// TwinCAT 3 PLC project PLC
// ProgramVersion: 3.1.4024.0
// libraries:
//   Tc2_ControllerToolbox, * (Beckhoff Automation GmbH)
//   Tc2_Standard, * (Beckhoff Automation GmbH)
//   Tc2_System, * (Beckhoff Automation GmbH)
//   Tc3_Module, * (Beckhoff Automation GmbH)
//   TcUnit, * (www.tcunit.org)
// project tree:
//   / PlcTask.TcTTO
//   POUs/3DOF robot/ FB_Clamp_INT.TcPOU, FB_RC_Servo.TcPOU, FB_Sequence_Executor.TcPOU, FB_Sequence_Recorder.TcPOU
//   POUs/3DOF robot/TEST/ FB_Clamp_INT_Test.TcPOU, FB_RC_Servo_Test.TcPOU, FB_Sequence_Recorder_Test.TcPOU, PRG_TEST_ThreeDOF_robot.TcPOU
//   POUs/Controller/ FB_Adaptive_PID_Controller.TcPOU, FB_Hysteresis.TcPOU, FB_PID_Controller.TcPOU
//   POUs/Controller/TEST/ PRG_Controller_TEST.TcPOU
//   POUs/Equipment simulation/ FB_MassSpringDamper.TcPOU, FB_Tank.TcPOU
//   POUs/Equipment simulation/TEST/ PRG_EquipmentSimulation_TEST.TcPOU
//   POUs/Filters/ FB_Filter_Floating_Average.TcPOU, FB_Filter_HighPass.TcPOU, FB_Filter_LowPass.TcPOU
//   POUs/Filters/TEST/ PRG_Filters_TEST.TcPOU
//   POUs/ Notes.TcPOU, Tips_and_tricks.TcPOU
//   POUs/Signal generators/ FB_Generator_PWM.TcPOU, FB_Generator_Random.TcPOU, FB_Generator_Sawtooth.TcPOU, FB_Generator_Sine.TcPOU, FB_Generator_Square.TcPOU, FB_Generator_Triangular.TcPOU
//   POUs/Signal generators/TEST/ PRG_SignalGenerators_TEST.TcPOU
//   POUs/Unit test example/ FB_Max_Value.TcPOU, FB_Max_Value_Test.TcPOU, PRG_TEST.TcPOU
// real-time tasks:
//   TASK PlcTask: cycle T#10ms, priority 20, ADS port 350

CONFIGURATION PLC
    RESOURCE PLC ON TwinCAT3
        TASK PlcTask(INTERVAL := T#10ms, PRIORITY := 20);
        PROGRAM PRG_TEST_ThreeDOF_robot WITH PlcTask : PRG_TEST_ThreeDOF_robot;
    END_RESOURCE
END_CONFIGURATION

// ---- POUs/3DOF robot/TEST/PRG_TEST_ThreeDOF_robot.TcPOU
PROGRAM PRG_TEST_ThreeDOF_robot
VAR
	fb_RC_Servo_Test : FB_RC_Servo_Test;
	fb_Sequence_Recorder : FB_Sequence_Recorder_Test;
	fb_Clamp_INT_Test : FB_Clamp_INT_Test;
END_VAR

TcUnit.RUN();

END_PROGRAM

// ---- POUs/3DOF robot/TEST/FB_RC_Servo_Test.TcPOU
FUNCTION_BLOCK FB_RC_Servo_Test EXTENDS TcUnit.FB_TestSuite

// SetpointReached();
// Stop();

METHOD PRIVATE OutputRamped
VAR_INPUT
END_VAR
END_METHOD

METHOD PRIVATE SetpointChanged
VAR_INPUT
END_VAR
END_METHOD

METHOD SetpointReached
VAR
	Servo : FB_RC_Servo;
	Setpoint : INT := 10;
	ExpectedSetpointReached : INT := 10;
	Result : INT;
END_VAR
TEST('TEST: Setpoint reached');

Servo(stop := FALSE,
	setpoint := Setpoint,
	rampSpeed := 10,
	trapezoidalProfileActive := FALSE,
	servoAngleMin := 0,
	servoAngleMax := 100,
	rampCycleTime := T#1MS,
	currentPositionSetpoint => Result);
	


AssertEquals(Expected := ExpectedSetpointReached,
	Actual := Servo.currentPositionSetpoint,
	Message := 'Expected value not reached');

TEST_FINISHED();
END_METHOD

METHOD PRIVATE StartingPosition
VAR_INPUT
END_VAR
END_METHOD

METHOD PRIVATE Stop
VAR
	stop : BOOL;
	init1 : BOOL := TRUE;
	init2 : BOOL := TRUE;
	init3 : BOOL := TRUE;
	intermediateVal1 : INT;
	intermediateVal2 : INT;
	valuesAreEqualAndNotZero : BOOL := FALSE;
	startValue : INT := 0;
	setpoint : INT := 10000;
	minValue : INT := 0;
	maxValue : INT := 10000;
	cycleTime : TIME := T#1MS;
	rampSpeed : INT := 20;
	FB_Servo: FB_RC_Servo;
	timer1: TON;
	timer2: TON;
	ExpectedValue : BOOL := TRUE;
END_VAR
IF init1 THEN
	stop := FALSE;
	init1 := FALSE;
END_IF;

timer1(IN:= TRUE, PT:= T#1000S, Q=> , ET=> );
timer2(IN:= TRUE, PT:= T#1000S, Q=> , ET=> );

FB_Servo(
	stop:= stop, 
	setpoint:= setpoint, 
	rampSpeed:= rampSpeed, 
	trapezoidalProfileActive:= FALSE, 
	servoAngleMin:= minValue, 
	servoAngleMax:= maxValue, 
	rampCycleTime:= cycleTime, 
	rampStartPos:= startValue, 
	currentPositionSetpoint=> , 
	error=> );

IF timer1.ET > T#1S AND init2 THEN
	stop := TRUE;
	intermediateVal1 := FB_Servo.currentPositionSetpoint;
	init2 := FALSE;
END_IF

IF timer2.ET > T#2S AND init3 THEN
	IF intermediateVal1 = intermediateVal2 AND intermediateVal1 <> 0 THEN
		valuesAreEqualAndNotZero := TRUE;
	END_IF
END_IF

AssertEquals(
Expected:= ExpectedValue,
 Actual:= valuesAreEqualAndNotZero,
 Message:= 'Ramp was not stopped or value was not ramped');
END_METHOD

METHOD PRIVATE Trapezoidal
VAR_INPUT
END_VAR
END_METHOD

END_FUNCTION_BLOCK

// ---- POUs/3DOF robot/FB_RC_Servo.TcPOU
FUNCTION_BLOCK FB_RC_Servo
VAR_INPUT
	stop : BOOL; // Stops motor at current position
	setpoint : INT; // Angle to reach
	rampSpeed : REAL; // Speed setpoint for servo angle
	trapezoidalProfileActive : BOOL; // Smooths speed of servo at start and end of movement
	servoAngleMin : INT; // Lower limit of function block output angle
	servoAngleMax : INT; // Upper limit of function block output angle
	rampCycleTime : TIME; // Set rampCycleTime to the same as the task sycle time
	rampStartPos : INT; // Starting position
END_VAR
VAR_OUTPUT
	currentPositionSetpoint : INT; // The actual output of function block
	error : STRING; // Error output for debug
END_VAR
VAR
	ramp : FB_CTRL_RAMP_GENERATOR;
	rampParameters : ST_CTRL_RAMP_GENERATOR_PARAMS;
END_VAR

rampParameters.fVeloNeg := rampSpeed;
rampParameters.fVeloPos := rampSpeed;
rampParameters.tCtrlCycleTime := rampCycleTime;
rampParameters.tTaskCycleTime := rampCycleTime;
ramp.fStart := rampStartPos;
ramp.fTarget := setpoint;

IF stop THEN
	ramp.bEnable := FALSE;
ELSE
	ramp.bEnable := TRUE;
END_IF

ramp(stParams := rampParameters);

END_FUNCTION_BLOCK

// ---- POUs/3DOF robot/FB_Sequence_Recorder.TcPOU
FUNCTION_BLOCK FB_Sequence_Recorder
VAR_INPUT
	inputBase : INT; // Base angle to be recorded
	inputShoulder : INT; // Shoulder angle to be recorded
	inputElbow : INT; // Elbow angle to be recorded
	recordPosition : BOOL; // Toggle to record current Base, Shoulder, and Elbow angles
	returnPositionAtIndex : INT; // outputBase, outputShoulder, and outputElbow are returned based on this value and recorded positions
	deletePositions : BOOL; // If true, all recorded values will be deleted
END_VAR
VAR_OUTPUT
	outputBase : INT; // Base angle returned based on returnPositonAtIndex
	outputShoulder : INT; // Shoulder angle returned based on returnPositonAtIndex
	outputElbow : INT; // Elbow angle returned based on returnPositonAtIndex
	numberRecordedPositions : INT; // Returns how many positions are saved
	ERROR_arrayFull : BOOL; // Returns true internal storage is full
	ERROR_duplicateValue : BOOL; // Returns true if two duplicate arm positions are attempted recorded simultanously
END_VAR
VAR
	currentIndex : INT := 0;
	basePositions : ARRAY[0..9] OF INT;
	shoulderPositions : ARRAY[0..9] OF INT;
	elbowPositions : ARRAY[0..9] OF INT;
	i : INT;
END_VAR

(* Handle deletion of all positions *)
IF deletePositions THEN
    FOR i := 0 TO 9 DO
        basePositions[i] := 0;
        shoulderPositions[i] := 0;
        elbowPositions[i] := 0;
    END_FOR
    numberRecordedPositions := 0;
    currentIndex := 0;
ELSE
    (* Ensure we do not exceed the array bounds *)
    IF currentIndex >= 10 THEN
        ERROR_arrayFull := TRUE;
    ELSE
        ERROR_arrayFull := FALSE;
        
        (* Check for duplicate only if at least one position is recorded *)
        IF recordPosition AND currentIndex > 0 THEN
            IF basePositions[currentIndex - 1] = inputBase AND 
               shoulderPositions[currentIndex - 1] = inputShoulder AND 
               elbowPositions[currentIndex - 1] = inputElbow THEN
                ERROR_duplicateValue := TRUE;
            ELSE
                ERROR_duplicateValue := FALSE;
            END_IF
        END_IF

        (* Record position if not a duplicate and space is available *)
        IF recordPosition AND NOT ERROR_duplicateValue AND NOT ERROR_arrayFull THEN
            basePositions[currentIndex] := inputBase;
            shoulderPositions[currentIndex] := inputShoulder;
            elbowPositions[currentIndex] := inputElbow;
            currentIndex := currentIndex + 1;
        END_IF
    END_IF

    (* Update the number of recorded positions *)
    numberRecordedPositions := currentIndex;
END_IF;

(* Return recorded position based on the requested index, with bounds check *)
IF returnPositionAtIndex >= 0 AND returnPositionAtIndex < currentIndex THEN
    outputBase := basePositions[returnPositionAtIndex];
    outputShoulder := shoulderPositions[returnPositionAtIndex];
    outputElbow := elbowPositions[returnPositionAtIndex];
ELSE
    outputBase := 0;
    outputShoulder := 0;
    outputElbow := 0;
END_IF;

END_FUNCTION_BLOCK

// ---- POUs/3DOF robot/TEST/FB_Sequence_Recorder_Test.TcPOU
FUNCTION_BLOCK FB_Sequence_Recorder_Test EXTENDS TcUnit.FB_TestSuite

AddOnePosition();
AddTwoPositions();
ClearPositions();
AddTwoClearAddOne();
TryAddDuplicatePosition();
NumberOfPositionsStored();
ZeroPositionsStored();
ArrayFull();

METHOD AddOnePosition
VAR
	inputBaseAngle : INT := 123;
	inputShoulderAngle : INT := 123;
	inputElbowAngle : INT := 123;
	expectedBaseAngle : INT := 123;
	actualBaseAngle : INT;
	FB_Seq_Rec: FB_Sequence_Recorder;
	recordPosition : BOOL := TRUE;
END_VAR
TEST('TEST: Add one position');

FB_Seq_Rec(
	inputBase:= inputBaseAngle, 
	inputShoulder:= inputShoulderAngle, 
	inputElbow:= inputElbowAngle, 
	recordPosition:= recordPosition, 
	returnPositionAtIndex:= 0, 
	deletePositions:= FALSE, 
	outputBase=> actualBaseAngle, 
	outputShoulder=> , 
	outputElbow=> , 
	numberRecordedPositions=> , 
	ERROR_arrayFull=> );

IF recordPosition THEN
	recordPosition := FALSE;
END_IF

AssertEquals(Expected := expectedBaseAngle,
	Actual := actualBaseAngle,
	Message := 'Position 1 was not recorded');
	
TEST_FINISHED();
END_METHOD

METHOD AddTwoClearAddOne
VAR
	inputBaseAngle1 : INT := 123;
	inputShoulderAngle1 : INT := 123;
	inputElbowAngle1 : INT := 123;
	expectedBaseAngle1 : INT := 123;
	inputBaseAngle2 : INT := 234;
	inputShoulderAngle2 : INT := 234;
	inputElbowAngle2 : INT := 234;
	expectedShoulderAngle2 : INT := 234;
	actualShoulderAngle1 : INT;
	actualShoulderAngle2 : INT;
	FB_Seq_Rec: FB_Sequence_Recorder;
	recordPosition : BOOL := TRUE;
	delete : BOOL := FALSE;
END_VAR
TEST('TEST: Add two, delete, then add one position');

FB_Seq_Rec(
	inputBase:= inputBaseAngle1, 
	inputShoulder:= inputShoulderAngle1, 
	inputElbow:= inputElbowAngle1, 
	recordPosition:= recordPosition, 
	returnPositionAtIndex:= 0, 
	deletePositions:= delete, 
	outputBase=> actualShoulderAngle1, 
	outputShoulder=> , 
	outputElbow=> , 
	numberRecordedPositions=> , 
	ERROR_arrayFull=> );
	
FB_Seq_Rec(
	inputBase:= inputBaseAngle2, 
	inputShoulder:= inputShoulderAngle2, 
	inputElbow:= inputElbowAngle2, 
	recordPosition:= recordPosition, 
	returnPositionAtIndex:= 1, 
	deletePositions:= delete, 
	outputBase=> , 
	outputShoulder=> actualShoulderAngle2, 
	outputElbow=> , 
	numberRecordedPositions=> , 
	ERROR_arrayFull=> );

delete := TRUE;
recordPosition := FALSE;

FB_Seq_Rec(
	inputBase:= inputBaseAngle2, 
	inputShoulder:= inputShoulderAngle2, 
	inputElbow:= inputElbowAngle2, 
	recordPosition:= recordPosition, 
	returnPositionAtIndex:= 1, 
	deletePositions:= delete, 
	outputBase=> , 
	outputShoulder=> actualShoulderAngle2, 
	outputElbow=> , 
	numberRecordedPositions=> , 
	ERROR_arrayFull=> );

delete := FALSE;
recordPosition := TRUE;


FB_Seq_Rec(
	inputBase:= inputBaseAngle2, 
	inputShoulder:= inputShoulderAngle2, 
	inputElbow:= inputElbowAngle2, 
	recordPosition:= recordPosition, 
	returnPositionAtIndex:= 0, 
	deletePositions:= delete, 
	outputBase=> , 
	outputShoulder=> actualShoulderAngle2, 
	outputElbow=> , 
	numberRecordedPositions=> , 
	ERROR_arrayFull=> );	

AssertEquals(Expected := expectedShoulderAngle2,
	Actual := actualShoulderAngle2,
	Message := 'Wrong value returned');
	
TEST_FINISHED();
END_METHOD

METHOD AddTwoPositions
VAR
	inputBaseAngle1 : INT := 123;
	inputShoulderAngle1 : INT := 123;
	inputElbowAngle1 : INT := 123;
	expectedBaseAngle1 : INT := 123;
	inputBaseAngle2 : INT := 234;
	inputShoulderAngle2 : INT := 234;
	inputElbowAngle2 : INT := 234;
	expectedShoulderAngle2 : INT := 234;
	actualShoulderAngle1 : INT;
	actualShoulderAngle2 : INT;
	FB_Seq_Rec: FB_Sequence_Recorder;
	recordPosition : BOOL := TRUE;
END_VAR
TEST('TEST: Add two positions');

FB_Seq_Rec(
	inputBase:= inputBaseAngle1, 
	inputShoulder:= inputShoulderAngle1, 
	inputElbow:= inputElbowAngle1, 
	recordPosition:= recordPosition, 
	returnPositionAtIndex:= 0, 
	deletePositions:= FALSE, 
	outputBase=> actualShoulderAngle1, 
	outputShoulder=> , 
	outputElbow=> , 
	numberRecordedPositions=> , 
	ERROR_arrayFull=> );
	
FB_Seq_Rec(
	inputBase:= inputBaseAngle2, 
	inputShoulder:= inputShoulderAngle2, 
	inputElbow:= inputElbowAngle2, 
	recordPosition:= recordPosition, 
	returnPositionAtIndex:= 1, 
	deletePositions:= FALSE, 
	outputBase=> , 
	outputShoulder=> actualShoulderAngle2, 
	outputElbow=> , 
	numberRecordedPositions=> , 
	ERROR_arrayFull=> );

IF recordPosition THEN
	recordPosition := FALSE;
END_IF

AssertEquals(Expected := expectedShoulderAngle2,
	Actual := actualShoulderAngle2,
	Message := 'Position 2 was not recorded');
	
TEST_FINISHED();
END_METHOD

METHOD ArrayFull
VAR
	expectedFeedback : BOOL := TRUE;
	actualFeedback : BOOL;
	FB_Seq_Rec: FB_Sequence_Recorder;
	recordPosition : BOOL := TRUE;
END_VAR
TEST('TEST: Array full');

FB_Seq_Rec(
	inputBase:= 1, 
	inputShoulder:= 0, 
	inputElbow:= 0, 
	recordPosition:= recordPosition, 
	returnPositionAtIndex:= 0, 
	deletePositions:= FALSE, 
	outputBase=> , 
	outputShoulder=> , 
	outputElbow=> , 
	numberRecordedPositions=> , 
	ERROR_arrayFull=> actualFeedback);
	
FB_Seq_Rec(
	inputBase:= 2, 
	inputShoulder:= 0, 
	inputElbow:= 0, 
	recordPosition:= recordPosition, 
	returnPositionAtIndex:= 0, 
	deletePositions:= FALSE, 
	outputBase=> , 
	outputShoulder=> , 
	outputElbow=> , 
	numberRecordedPositions=> , 
	ERROR_arrayFull=> actualFeedback);
	
FB_Seq_Rec(
	inputBase:= 3, 
	inputShoulder:= 0, 
	inputElbow:= 0, 
	recordPosition:= recordPosition, 
	returnPositionAtIndex:= 0, 
	deletePositions:= FALSE, 
	outputBase=> , 
	outputShoulder=> , 
	outputElbow=> , 
	numberRecordedPositions=> , 
	ERROR_arrayFull=> actualFeedback);
	
FB_Seq_Rec(
	inputBase:= 4, 
	inputShoulder:= 0, 
	inputElbow:= 0, 
	recordPosition:= recordPosition, 
	returnPositionAtIndex:= 0, 
	deletePositions:= FALSE, 
	outputBase=> , 
	outputShoulder=> , 
	outputElbow=> , 
	numberRecordedPositions=> , 
	ERROR_arrayFull=> actualFeedback);
	
FB_Seq_Rec(
	inputBase:= 5, 
	inputShoulder:= 0, 
	inputElbow:= 0, 
	recordPosition:= recordPosition, 
	returnPositionAtIndex:= 0, 
	deletePositions:= FALSE, 
	outputBase=> , 
	outputShoulder=> , 
	outputElbow=> , 
	numberRecordedPositions=> , 
	ERROR_arrayFull=> actualFeedback);
	
FB_Seq_Rec(
	inputBase:= 6, 
	inputShoulder:= 0, 
	inputElbow:= 0, 
	recordPosition:= recordPosition, 
	returnPositionAtIndex:= 0, 
	deletePositions:= FALSE, 
	outputBase=> , 
	outputShoulder=> , 
	outputElbow=> , 
	numberRecordedPositions=> , 
	ERROR_arrayFull=> actualFeedback);
	
FB_Seq_Rec(
	inputBase:= 7, 
	inputShoulder:= 0, 
	inputElbow:= 0, 
	recordPosition:= recordPosition, 
	returnPositionAtIndex:= 0, 
	deletePositions:= FALSE, 
	outputBase=> , 
	outputShoulder=> , 
	outputElbow=> , 
	numberRecordedPositions=> , 
	ERROR_arrayFull=> actualFeedback);
	
FB_Seq_Rec(
	inputBase:= 8, 
	inputShoulder:= 0, 
	inputElbow:= 0, 
	recordPosition:= recordPosition, 
	returnPositionAtIndex:= 0, 
	deletePositions:= FALSE, 
	outputBase=> , 
	outputShoulder=> , 
	outputElbow=> , 
	numberRecordedPositions=> , 
	ERROR_arrayFull=> actualFeedback);
	
FB_Seq_Rec(
	inputBase:= 9, 
	inputShoulder:= 0, 
	inputElbow:= 0, 
	recordPosition:= recordPosition, 
	returnPositionAtIndex:= 0, 
	deletePositions:= FALSE, 
	outputBase=> , 
	outputShoulder=> , 
	outputElbow=> , 
	numberRecordedPositions=> , 
	ERROR_arrayFull=> actualFeedback);
	
FB_Seq_Rec(
	inputBase:= 10, 
	inputShoulder:= 0, 
	inputElbow:= 0, 
	recordPosition:= recordPosition, 
	returnPositionAtIndex:= 0, 
	deletePositions:= FALSE, 
	outputBase=> , 
	outputShoulder=> , 
	outputElbow=> , 
	numberRecordedPositions=> , 
	ERROR_arrayFull=> actualFeedback);
	
FB_Seq_Rec(
	inputBase:= 11, 
	inputShoulder:= 0, 
	inputElbow:= 0, 
	recordPosition:= recordPosition, 
	returnPositionAtIndex:= 0, 
	deletePositions:= FALSE, 
	outputBase=> , 
	outputShoulder=> , 
	outputElbow=> , 
	numberRecordedPositions=> , 
	ERROR_arrayFull=> actualFeedback);


AssertEquals(Expected := expectedFeedback,
	Actual := actualFeedback,
	Message := 'Alarm indicating full array not activated');
	
TEST_FINISHED();
END_METHOD

METHOD ClearPositions : BOOL
VAR
	inputBaseAngle1 : INT := 123;
	inputShoulderAngle1 : INT := 123;
	inputElbowAngle1 : INT := 123;
	expectedBaseAngle1 : INT := 123;
	inputBaseAngle2 : INT := 234;
	inputShoulderAngle2 : INT := 234;
	inputElbowAngle2 : INT := 234;
	expectedShoulderAngle2 : INT := 0;
	actualShoulderAngle1 : INT;
	actualShoulderAngle2 : INT;
	FB_Seq_Rec: FB_Sequence_Recorder;
	recordPosition : BOOL := TRUE;
	delete : BOOL := FALSE;
END_VAR
TEST('TEST: Clear positions');

FB_Seq_Rec(
	inputBase:= inputBaseAngle1, 
	inputShoulder:= inputShoulderAngle1, 
	inputElbow:= inputElbowAngle1, 
	recordPosition:= recordPosition, 
	returnPositionAtIndex:= 0, 
	deletePositions:= FALSE, 
	outputBase=> actualShoulderAngle1, 
	outputShoulder=> , 
	outputElbow=> , 
	numberRecordedPositions=> , 
	ERROR_arrayFull=> );
	
FB_Seq_Rec(
	inputBase:= inputBaseAngle2, 
	inputShoulder:= inputShoulderAngle2, 
	inputElbow:= inputElbowAngle2, 
	recordPosition:= recordPosition, 
	returnPositionAtIndex:= 1, 
	deletePositions:= delete, 
	outputBase=> , 
	outputShoulder=> actualShoulderAngle2, 
	outputElbow=> , 
	numberRecordedPositions=> , 
	ERROR_arrayFull=> );

IF recordPosition THEN
	recordPosition := FALSE;
END_IF

delete := TRUE;

FB_Seq_Rec(
	inputBase:= inputBaseAngle2, 
	inputShoulder:= inputShoulderAngle2, 
	inputElbow:= inputElbowAngle2, 
	recordPosition:= recordPosition, 
	returnPositionAtIndex:= 1, 
	deletePositions:= delete, 
	outputBase=> , 
	outputShoulder=> actualShoulderAngle2, 
	outputElbow=> , 
	numberRecordedPositions=> , 
	ERROR_arrayFull=> );

AssertEquals(Expected := expectedShoulderAngle2,
	Actual := actualShoulderAngle2,
	Message := 'Positions were not deleted');
	
TEST_FINISHED();
END_METHOD

METHOD ErrorIndexOutOfBounds
VAR_INPUT
END_VAR
// Should not be able to input values larger than 9, as it is only possible to store 10 positions in the array (0-9)
//
END_METHOD

METHOD NumberOfPositionsStored : REFERENCE TO FB_Test
VAR
	FB_Seq_Rec: FB_Sequence_Recorder;
	expectedNumberOfPositionsStored : INT := 5;
	actualNumberOfPositionsStored : INT;
END_VAR
TEST('Return number of positions stored');

FB_Seq_Rec(
	inputBase:= 0, 
	inputShoulder:= 0, 
	inputElbow:= 0, 
	recordPosition:= TRUE, 
	returnPositionAtIndex:= 0, 
	deletePositions:= FALSE, 
	outputBase=> , 
	outputShoulder=> , 
	outputElbow=> , 
	numberRecordedPositions=> actualNumberOfPositionsStored, 
	ERROR_arrayFull=> );
	
FB_Seq_Rec(
	inputBase:= 1, 
	inputShoulder:= 0, 
	inputElbow:= 0, 
	recordPosition:= TRUE, 
	returnPositionAtIndex:= 0, 
	deletePositions:= FALSE, 
	outputBase=> , 
	outputShoulder=> , 
	outputElbow=> , 
	numberRecordedPositions=> actualNumberOfPositionsStored, 
	ERROR_arrayFull=> );
	
FB_Seq_Rec(
	inputBase:= 0, 
	inputShoulder:= 0, 
	inputElbow:= 0, 
	recordPosition:= TRUE, 
	returnPositionAtIndex:= 0, 
	deletePositions:= FALSE, 
	outputBase=> , 
	outputShoulder=> , 
	outputElbow=> , 
	numberRecordedPositions=> actualNumberOfPositionsStored, 
	ERROR_arrayFull=> );

// DELETE
FB_Seq_Rec(
	inputBase:= 1, 
	inputShoulder:= 1, 
	inputElbow:= 1, 
	recordPosition:= FALSE, 
	returnPositionAtIndex:= 0, 
	deletePositions:= TRUE, 
	outputBase=> , 
	outputShoulder=> , 
	outputElbow=> , 
	numberRecordedPositions=> actualNumberOfPositionsStored, 
	ERROR_arrayFull=> );
	
FB_Seq_Rec(
	inputBase:= 2, 
	inputShoulder:= 2, 
	inputElbow:= 2, 
	recordPosition:= TRUE, 
	returnPositionAtIndex:= 0, 
	deletePositions:= FALSE, 
	outputBase=> , 
	outputShoulder=> , 
	outputElbow=> , 
	numberRecordedPositions=> actualNumberOfPositionsStored, 
	ERROR_arrayFull=> );
	
FB_Seq_Rec(
	inputBase:= 3, 
	inputShoulder:= 3, 
	inputElbow:= 3, 
	recordPosition:= TRUE, 
	returnPositionAtIndex:= 0, 
	deletePositions:= FALSE, 
	outputBase=> , 
	outputShoulder=> , 
	outputElbow=> , 
	numberRecordedPositions=> actualNumberOfPositionsStored, 
	ERROR_arrayFull=> );
	
FB_Seq_Rec(
	inputBase:= 4, 
	inputShoulder:= 4, 
	inputElbow:= 4, 
	recordPosition:= TRUE, 
	returnPositionAtIndex:= 0, 
	deletePositions:= FALSE, 
	outputBase=> , 
	outputShoulder=> , 
	outputElbow=> , 
	numberRecordedPositions=> actualNumberOfPositionsStored, 
	ERROR_arrayFull=> );
	
FB_Seq_Rec(
	inputBase:= 5, 
	inputShoulder:= 5, 
	inputElbow:= 5, 
	recordPosition:= TRUE, 
	returnPositionAtIndex:= 0, 
	deletePositions:= FALSE, 
	outputBase=> , 
	outputShoulder=> , 
	outputElbow=> , 
	numberRecordedPositions=> actualNumberOfPositionsStored, 
	ERROR_arrayFull=> );
	
FB_Seq_Rec(
	inputBase:= 6, 
	inputShoulder:= 6, 
	inputElbow:= 6, 
	recordPosition:= TRUE, 
	returnPositionAtIndex:= 0, 
	deletePositions:= FALSE, 
	outputBase=> , 
	outputShoulder=> , 
	outputElbow=> , 
	numberRecordedPositions=> actualNumberOfPositionsStored, 
	ERROR_arrayFull=> );
	
AssertEquals(Expected := expectedNumberOfPositionsStored,
	Actual := actualNumberOfPositionsStored,
	Message := 'Wrong number of positions stored returned');
	
TEST_FINISHED();
END_METHOD

METHOD TryAddDuplicatePosition
VAR
	inputBaseAngle1 : INT := 123;
	inputShoulderAngle1 : INT := 123;
	inputElbowAngle1 : INT := 123;
	expectedBaseAngle1 : INT := 0;
	inputBaseAngle2 : INT := 0;
	inputShoulderAngle2 : INT := 0;
	inputElbowAngle2 : INT := 0;
	expectedResult : BOOL := FALSE;
	actualBaseAngle1 : INT;
	actualShoulderAngle1 : INT;
	actualElbowAngle1 : INT;
	actualBaseAngle2 : INT;
	actualShoulderAngle2 : INT;
	actualElbowAngle2 : INT;
	FB_Seq_Rec: FB_Sequence_Recorder;
	recordPosition : BOOL := TRUE;
	arePositionsDuplicate: BOOL := FALSE;
END_VAR
TEST('TEST: Try add duplicate positions');

FB_Seq_Rec(
	inputBase:= inputBaseAngle1, 
	inputShoulder:= inputShoulderAngle1, 
	inputElbow:= inputElbowAngle1, 
	recordPosition:= recordPosition, 
	returnPositionAtIndex:= 0, 
	deletePositions:= FALSE, 
	outputBase=> actualBaseAngle1, 
	outputShoulder=> actualShoulderAngle1, 
	outputElbow=> actualElbowAngle1, 
	numberRecordedPositions=> , 
	ERROR_arrayFull=> );
	
FB_Seq_Rec(
	inputBase:= inputBaseAngle2, 
	inputShoulder:= inputShoulderAngle2, 
	inputElbow:= inputElbowAngle2, 
	recordPosition:= recordPosition, 
	returnPositionAtIndex:= 1, 
	deletePositions:= FALSE, 
	outputBase=> actualBaseAngle2, 
	outputShoulder=> actualShoulderAngle2, 
	outputElbow=> actualElbowAngle2, 
	numberRecordedPositions=> , 
	ERROR_arrayFull=> );
	
IF (actualBaseAngle1 = actualBaseAngle2) AND (actualShoulderAngle1 = actualShoulderAngle2) AND (actualElbowAngle1 = actualElbowAngle1) THEN
	arePositionsDuplicate := TRUE;
END_IF

AssertEquals(Expected := expectedResult,
	Actual := arePositionsDuplicate,
	Message := 'Not allowed to add duplicate values!');
	
TEST_FINISHED();
END_METHOD

METHOD ZeroPositionsStored
VAR
	inputBaseAngle : INT := 123;
	inputShoulderAngle : INT := 123;
	inputElbowAngle : INT := 123;
	expectedNumberOfPositionsStored : INT := 0;
	actualNumberOfPositionsStored : INT;
	FB_Seq_Rec: FB_Sequence_Recorder;
	recordPosition : BOOL := FALSE;
END_VAR
TEST('TEST: Zero positions added');

FB_Seq_Rec(
	inputBase:= inputBaseAngle, 
	inputShoulder:= inputShoulderAngle, 
	inputElbow:= inputElbowAngle, 
	recordPosition:= recordPosition, 
	returnPositionAtIndex:= 0, 
	deletePositions:= FALSE, 
	outputBase=> , 
	outputShoulder=> , 
	outputElbow=> , 
	numberRecordedPositions=> actualNumberOfPositionsStored, 
	ERROR_arrayFull=> );


AssertEquals(Expected := expectedNumberOfPositionsStored,
	Actual := actualNumberOfPositionsStored,
	Message := 'There are no positions recorrded');
	
TEST_FINISHED();
END_METHOD

END_FUNCTION_BLOCK

// ---- POUs/3DOF robot/TEST/FB_Clamp_INT_Test.TcPOU
FUNCTION_BLOCK FB_Clamp_INT_Test  EXTENDS TcUnit.FB_TestSuite

OutOfBoundsUpper();
OutOfBoundsLower();
ValidInput();

METHOD OutOfBoundsLower : REFERENCE TO FB_Test
VAR
	Input : INT := -100;
	Upper : INT := 180;
	Lower : INT := 0;
	ExpectedOutput : INT := 0;
	ActualOutput : INT;
	Clamp: FB_Clamp_INT;
END_VAR
TEST('TEST: Out of bounds lower');

Clamp(
	Input:= Input, 
	UpperLimit:= Upper, 
	LowerLimit:= Lower, 
	Output=> ActualOutput, 
	OutOfBounds=> );

	
AssertEquals(Expected := ExpectedOutput,
	Actual := ActualOutput,
	Message := 'Not expected output');

TEST_FINISHED();
END_METHOD

METHOD OutOfBoundsUpper
VAR
	Input : INT := 200;
	Upper : INT := 180;
	Lower : INT := 0;
	ExpectedOutput : INT := 180;
	ActualOutput : INT;
	Clamp: FB_Clamp_INT;
END_VAR
TEST('TEST: Out of bounds upper');

Clamp(
	Input:= Input, 
	UpperLimit:= Upper, 
	LowerLimit:= Lower, 
	Output=> ActualOutput, 
	OutOfBounds=> );

	
AssertEquals(Expected := ExpectedOutput,
	Actual := ActualOutput,
	Message := 'Not expected output');

TEST_FINISHED();
END_METHOD

METHOD ValidInput
VAR
	Input : INT := 150;
	Upper : INT := 180;
	Lower : INT := 0;
	ExpectedOutput : INT := 150;
	ActualOutput : INT;
	Clamp: FB_Clamp_INT;
END_VAR
TEST('TEST: Valid input');

Clamp(
	Input:= Input, 
	UpperLimit:= Upper, 
	LowerLimit:= Lower, 
	Output=> ActualOutput, 
	OutOfBounds=> );

	
AssertEquals(Expected := ExpectedOutput,
	Actual := ActualOutput,
	Message := 'Not expected output');

TEST_FINISHED();
END_METHOD

END_FUNCTION_BLOCK

// ---- POUs/3DOF robot/FB_Clamp_INT.TcPOU
FUNCTION_BLOCK FB_Clamp_INT
VAR_INPUT
	Input : INT;
	UpperLimit :INT;
	LowerLimit : INT;
END_VAR
VAR_OUTPUT
	Output : INT;
	OutOfBounds : BOOL;
END_VAR

IF Input > UpperLimit THEN
	Output := UpperLimit;
ELSIF Input < LowerLimit THEN
	Output := LowerLimit;
ELSIF Input < UpperLimit AND Input > LowerLimit THEN
	Output := Input;
END_IF

END_FUNCTION_BLOCK

// ---- POUs/3DOF robot/FB_Sequence_Executor.TcPOU
FUNCTION_BLOCK FB_Sequence_Executor
VAR_INPUT
	enableSequence : BOOL; // If true, output angles will be ramped. If false, output angles will be freezed
	baseSetpoint : INT; // Base angle setpoint
	shoulderSetpoint : INT; // Shoulder angle setpoint
	elbowSetpoint : INT; // Elbow angle setpoint
	enableLoop : BOOL; // If true, sequence will start over when finished
	speed : INT; // Speed of servos
	numberPositionsRecorded : INT; // Will be used to keep track on when to loop back to first position
	restart : INT; // Will start sequence from first recorded position
END_VAR
VAR_OUTPUT
	currentBaseAngleSetpoint : INT; // Ramped setpoint to be sent to base servo
	currentShoulderAngleSetpoint : INT; // Ramped setpoint to be sent to shoulder servo
	currentElbowAngleSetpoint : INT; // Ramped setpoint to be sent to elbow servo
	finalPosReached : BOOL; // When sequence is done, this variable will be true
	selectIndex : INT; // This variable will be incremented when intermediate positions have been reached
END_VAR
VAR
	FB_BaseServo : FB_RC_Servo; // Base servo function block
	FB_ShoulderServo : FB_RC_Servo; // Shoulder servo function block
	FB_ElbowServo : FB_RC_Servo; // Elbow servo function block
END_VAR

END_FUNCTION_BLOCK

// ---- POUs/Controller/FB_Adaptive_PID_Controller.TcPOU
PROGRAM FB_Adaptive_PID_Controller
VAR
END_VAR

END_PROGRAM

// ---- POUs/Controller/FB_Hysteresis.TcPOU
FUNCTION_BLOCK FB_Hysteresis
VAR_INPUT
	setpoint : REAL;
	feedback : REAL;
	upperLimit : REAL;
	lowerLimit : REAL;
	controlSignalLow : REAL;
	controlSignalHigh : REAL;
END_VAR
VAR_OUTPUT
END_VAR
VAR_IN_OUT
	controlSignal : REAL;
END_VAR
VAR
END_VAR


IF feedback > lowerLimit THEN
	controlSignal := controlSignalHigh;
ELSE
	controlSignal := controlsignalHigh;
END_IF

END_FUNCTION_BLOCK

// ---- POUs/Controller/FB_PID_Controller.TcPOU
FUNCTION_BLOCK FB_PID_Controller
VAR_INPUT
	setpoint : REAL;
	feedback : REAL;
	KP : REAL;
	KI : REAL;
	KD : REAL;
END_VAR
VAR_OUTPUT
	controlSignal : REAL;
END_VAR
VAR
	currentError : REAL;
	accumulatedError : REAL;
	deltaError : REAL;
END_VAR

error := setpoint - feedback;

controlSignal := KP*error + KI*accumulatedError + KD*deltaError;

END_FUNCTION_BLOCK

// ---- POUs/Controller/TEST/PRG_Controller_TEST.TcPOU
PROGRAM PRG_Controller_TEST
VAR
END_VAR

END_PROGRAM

// ---- POUs/Equipment simulation/FB_MassSpringDamper.TcPOU
PROGRAM FB_MassSpringDamper
VAR
END_VAR

END_PROGRAM

// ---- POUs/Equipment simulation/FB_Tank.TcPOU
PROGRAM FB_Tank
VAR
END_VAR

END_PROGRAM

// ---- POUs/Equipment simulation/TEST/PRG_EquipmentSimulation_TEST.TcPOU
PROGRAM PRG_EquipmentSimulation_TEST
VAR
END_VAR

END_PROGRAM

// ---- POUs/Filters/FB_Filter_Floating_Average.TcPOU
FUNCTION_BLOCK FB_Filter_Floating_Average
VAR_INPUT
END_VAR
VAR_OUTPUT
END_VAR
VAR
END_VAR

END_FUNCTION_BLOCK

// ---- POUs/Filters/FB_Filter_HighPass.TcPOU
FUNCTION_BLOCK FB_Filter_HighPass
VAR_INPUT
END_VAR
VAR_OUTPUT
END_VAR
VAR
END_VAR

END_FUNCTION_BLOCK

// ---- POUs/Filters/FB_Filter_LowPass.TcPOU
FUNCTION_BLOCK FB_Filter_LowPass
VAR_INPUT
END_VAR
VAR_OUTPUT
END_VAR
VAR
END_VAR

END_FUNCTION_BLOCK

// ---- POUs/Filters/TEST/PRG_Filters_TEST.TcPOU
PROGRAM PRG_Filters_TEST
VAR
END_VAR

END_PROGRAM

// ---- POUs/Notes.TcPOU
PROGRAM Notes
VAR
END_VAR

// Write notes here

// Comment out

END_PROGRAM

// ---- POUs/Signal generators/FB_Generator_PWM.TcPOU
FUNCTION_BLOCK FB_Generator_PWM
VAR_INPUT
END_VAR
VAR_OUTPUT
END_VAR
VAR
END_VAR

END_FUNCTION_BLOCK

// ---- POUs/Signal generators/FB_Generator_Random.TcPOU
FUNCTION_BLOCK FB_Generator_Random
VAR_INPUT
END_VAR
VAR_OUTPUT
END_VAR
VAR
END_VAR

END_FUNCTION_BLOCK

// ---- POUs/Signal generators/FB_Generator_Sawtooth.TcPOU
FUNCTION_BLOCK FB_Generator_Sawtooth
VAR_INPUT
END_VAR
VAR_OUTPUT
END_VAR
VAR
END_VAR

END_FUNCTION_BLOCK

// ---- POUs/Signal generators/FB_Generator_Sine.TcPOU
FUNCTION_BLOCK FB_Generator_Sine
VAR_INPUT
END_VAR
VAR_OUTPUT
END_VAR
VAR
END_VAR

END_FUNCTION_BLOCK

// ---- POUs/Signal generators/FB_Generator_Square.TcPOU
FUNCTION_BLOCK FB_Generator_Square
VAR_INPUT
END_VAR
VAR_OUTPUT
END_VAR
VAR
END_VAR

END_FUNCTION_BLOCK

// ---- POUs/Signal generators/FB_Generator_Triangular.TcPOU
FUNCTION_BLOCK FB_Generator_Triangular
VAR_INPUT
END_VAR
VAR_OUTPUT
END_VAR
VAR
END_VAR

END_FUNCTION_BLOCK

// ---- POUs/Signal generators/TEST/PRG_SignalGenerators_TEST.TcPOU
PROGRAM PRG_SignalGenerators_TEST
VAR
END_VAR

END_PROGRAM

// ---- POUs/Tips_and_tricks.TcPOU
PROGRAM Tips_and_tricks
VAR
END_VAR

// Shortcuts

// Comment muliple lines of code: CTRL + K, CTRL + U
// Uncomment multiple lines of code : CTRL + K, CTRL + U

END_PROGRAM

// ---- POUs/Unit test example/FB_Max_Value.TcPOU
FUNCTION_BLOCK FB_Max_Value
VAR_INPUT
	value1 : LREAL;
	value2 : LREAL;
END_VAR
VAR_OUTPUT
	result : LREAL;
END_VAR

IF value1 >= value2 THEN
	result := value1;
ELSIF value1 <= value2 THEN
	result := value2;
END_IF

END_FUNCTION_BLOCK

// ---- POUs/Unit test example/FB_Max_Value_Test.TcPOU
FUNCTION_BLOCK FB_Max_Value_Test EXTENDS TcUnit.FB_TestSuite
VAR
END_VAR

FirstValueIsBiggest();
SecondValueIsBiggest();
ValuesAreEqual();

METHOD FirstValueIsBiggest
VAR
	Maximum : FB_Max_Value;
	Result: LREAL;
	ExpectedMax : LREAL := 3;
END_VAR
TEST('TEST: First Value Is Biggest');

Maximum(value1 := 3, value2 := 1, result => Result);

AssertEquals(Expected := ExpectedMax,
			Actual := Result,
			Message := 'Max value not found');

TEST_FINISHED();
END_METHOD

METHOD SecondValueIsBiggest
VAR
	Maximum : FB_Max_Value;
	Result : LREAL;
	ExpectedMax : LREAL := 9;
	
END_VAR
TEST('TEST: Second value is largest');

Maximum(value1 := 1, value2 := 9, result => Result);

AssertEquals(Expected := ExpectedMax,
			Actual := Result,
			Message := 'Largest value not found');

TEST_FINISHED();
END_METHOD

METHOD ValuesAreEqual
VAR
	Maximum : FB_Max_Value;
	Result : LREAL;
	ExpectedMax : LREAL := -999;
END_VAR
TEST('Checks output if both input values are the same');

Maximum(value1 := -999,
		value2 := -999,
		result => Result);

AssertEquals(Expected := ExpectedMax,
			Actual := Result,
			Message := 'Largest value not found');
			
TEST_FINISHED();
END_METHOD

END_FUNCTION_BLOCK

// ---- POUs/Unit test example/PRG_TEST.TcPOU
PROGRAM PRG_TEST
VAR
	fb_Max_Value_Test : FB_Max_Value_Test;
END_VAR

TcUnit.RUN();

END_PROGRAM
